PROGRAM POU_Saw
VAR
	start_timer :BOOL;
	timer : ton;
	timer1: ton;
	PT: INT;
END_VAR

END_PROGRAM

(* stored: Version 1.1.0.1, ProductVersion 3.1.4024.12
   POU POU_Saw: Id {20362c0f-2be3-4923-bb5c-847f6c28e7d5}, SpecialFunc None *)
